FUNCTION Convert_ULINT_TO_WORD : Hresult
VAR_INPUT
	in : ULINT;
	out : REFERENCE TO WORD;
END_VAR
VAR
	converted : WORD;
END_VAR

converted := ULINT_TO_WORD(in);

IF (WORD_TO_ULINT(converted) <> in) THEN
	Convert_ULINT_TO_WORD := INCOMPATIBLE;
	RETURN;
END_IF

out := converted;

END_FUNCTION

(* stored: Version 1.1.0.1, ProductVersion 3.1.4024.12
   POU Convert_ULINT_TO_WORD: Id {12fa1308-1e76-4c5a-a8ee-d8fac6cceac0}, SpecialFunc None *)
